Universal Robots PolyScope program: b_zback4.urp

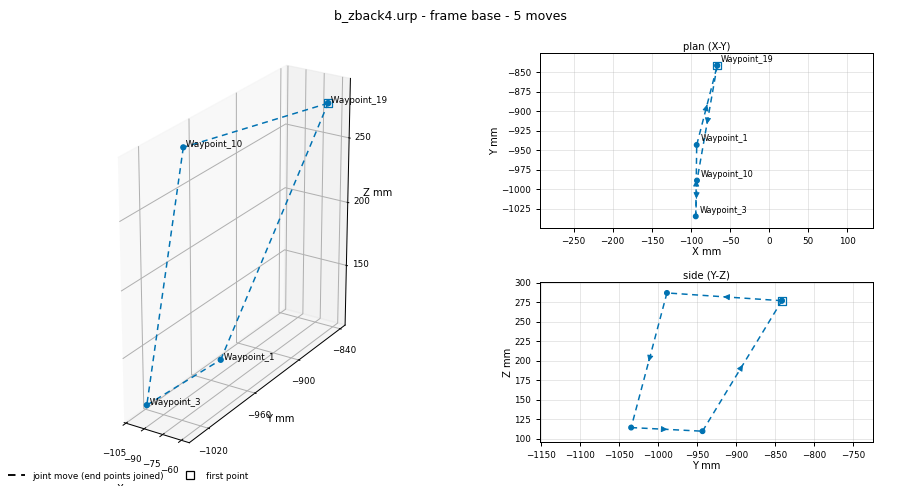
[picture p0: tool path of b_zback4.urp in frame base, 5 of 5 moves have a stored position in this frame; points joined in program order, loops and branches not executed]
Program b_zback4 (installation=default directory=/programs/Burkat_U_Plant createdIn=5.12.6.1102099 lastSavedIn=5.12.6.1102099 robotSerialNumber=20215500597)
Calibrated DH parameters: a=[0.000193, -0.066673, -0.391568, -0.000012, 0.00005, 0]; d=[0.162643, -472.05677, 465.132521, 7.058239, 0.099746, 0.099582]; alpha=[1.571116, 0.00089, 0.003862, 1.569269, -1.569248, 0]; deltaTheta=[0, -1.413394, 7.628392, 0.068187, 0, -0.000001]
Robot Program (runOnlyOnce=true)
  MoveJ speed 60 deg/s, acceleration 80 deg/s^2 (useActiveTCP=true) feature=Base
    Waypoint Waypoint_19: TCP in base x=-66.326 y=-841.615 z=276.687 mm, rx=1.6517 ry=-0.0259 rz=-0.093 rad; joints [71.48, -64.638, 86.648, -17.383, 75.945, -3.629] deg; TCP offset x=0 y=0 z=191.5 mm, rx=0 ry=0 rz=0 rad
    Waypoint Waypoint_10: TCP in base x=-92.228 y=-988.698 z=286.655 mm, rx=1.6465 ry=0.0332 rz=-0.0452 rad; joints [71.779, -43.319, 50.021, -2.274, 72.327, -4.08] deg
    Waypoint Waypoint_3: motionParameters(jointSpeed=0.349066 jointAcceleration=1.047198 cartesianSpeed=0.25 cartesianAcceleration=1.2); TCP in base x=-93.776 y=-1034.526 z=114.346 mm, rx=1.6139 ry=0.0476 rz=-0.0472 rad; joints [72.59, -28.312, 48.772, -17.976, 72.673, -4.058] deg
  URCap Gripper (Robotiq_Grippers, Robotiq Inc.) dataModel(position=0.0, force=29.019607843137255, speed=30.11764705882353, positionInDouble=0.0, forceInDouble=29.019607843137255, speedInDouble=30.11764705882353, slaveIds=[9], blocking=true)
  MoveJ speed 30 deg/s, acceleration 40 deg/s^2 (useActiveTCP=true) feature=Base
    Waypoint Waypoint_1: motionParameters(jointSpeed=0.087266 jointAcceleration=0.174533 cartesianSpeed=0.25 cartesianAcceleration=1.2); TCP in base x=-92.58 y=-943.208 z=109.706 mm, rx=1.5938 ry=0.0536 rz=-0.0777 rad; joints [70.625, -40.487, 74.961, -33.19, 71.628, -5.097] deg
    Waypoint Waypoint_19: TCP in base x=-66.326 y=-841.615 z=276.687 mm, rx=1.6517 ry=-0.0259 rz=-0.093 rad; joints [71.48, -64.638, 86.648, -17.383, 75.945, -3.629] deg
